SUBAPPLICATION Uebung_208_AX (* Interlock: ILOCK_FB_SR_AX (Zwei gegenseitig verriegelte Set-Dominante Latches via AX/AX2-Adapter) *)
  (* Standard: 61499-2; Description: Copyright (c) 2026 Meisterschulen am Ostbahnhof This program and the accompanying materials are made available under the terms of the Eclipse Public License 2.0 which is available at https://www.eclipse.org/legal/epl-2.0/ SPDX-License-Identifier: EPL-2.0 *)
  (* Version 1.0, 2026-05-07, Gemini CLI, Meisterschulen am Ostbahnhof, initial version using library block ILOCK_FB_SR_AX *)
  PACKAGE Uebungen;
  IMPORT logiBUS::io::DI::logiBUS_DI::Input_I1;
  IMPORT logiBUS::io::DI::logiBUS_DI::Input_I2;
  IMPORT logiBUS::io::DI::logiBUS_DI::Input_I3;
  IMPORT logiBUS::io::DI::logiBUS_DI::Input_I4;
  IMPORT logiBUS::io::DQ::logiBUS_DO::Output_Q1;
  IMPORT logiBUS::io::DQ::logiBUS_DO::Output_Q2;
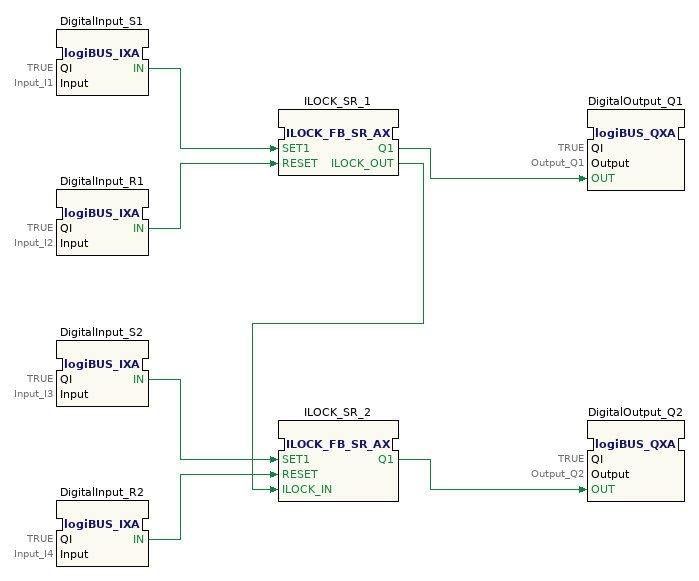
  FBS
    DigitalInput_S1 : logiBUS::io::DI::logiBUS_IXA(QI := TRUE, Input := Input_I1);
    DigitalInput_R1 : logiBUS::io::DI::logiBUS_IXA(QI := TRUE, Input := Input_I2);
    DigitalInput_S2 : logiBUS::io::DI::logiBUS_IXA(QI := TRUE, Input := Input_I3);
    DigitalInput_R2 : logiBUS::io::DI::logiBUS_IXA(QI := TRUE, Input := Input_I4);
    ILOCK_SR_1 : logiBUS::signalprocessing::interlock::ILOCK_FB_SR_AX;
    ILOCK_SR_2 : logiBUS::signalprocessing::interlock::ILOCK_FB_SR_AX;
    DigitalOutput_Q1 : logiBUS::io::DQ::logiBUS_QXA(QI := TRUE, Output := Output_Q1);
    DigitalOutput_Q2 : logiBUS::io::DQ::logiBUS_QXA(QI := TRUE, Output := Output_Q2);
  END_FBS
  ADAPTER_CONNECTIONS
    DigitalInput_S1.IN TO ILOCK_SR_1.SET1;
    DigitalInput_R1.IN TO ILOCK_SR_1.RESET;
    DigitalInput_S2.IN TO ILOCK_SR_2.SET1;
    DigitalInput_R2.IN TO ILOCK_SR_2.RESET;
    ILOCK_SR_1.Q1 TO DigitalOutput_Q1.OUT;
    ILOCK_SR_2.Q1 TO DigitalOutput_Q2.OUT;
    ILOCK_SR_1.ILOCK_OUT TO ILOCK_SR_2.ILOCK_IN;
  END_CONNECTIONS
END_SUBAPPLICATION
